// SIMATIC S7-200 project (STEP 7-Micro/WIN), CPU 226 REL 01.01

SYMBOL_TABLE USR1
Any_100ms_Timer  T38
END_SYMBOL_TABLE

SYMBOL_TABLE USS Protocol
USS_LOW_V        VD1000   // (DWORD) Enter the starting address for USS Protocol symbols here.
USS_HIGH_V       VD1004
USS_TIME_OUT     VW1008
USS_I_LINE       VW1010
USS_DAT_PTR0     VD1012
USS_ACT_DRV0     VD1016
USS_CUR_DRV0     VD1020
USS_P0           V1024.0
USS_REQ_SNT0     V1024.1
USS_RETRY_P0     VB1025
USS_ERR_CODE     VB1026
USS_CS_D0        VD1027
USS_CS_W0        VW1027
USS_CS_W2        VW1029
USS_CS_B0        VB1027
USS_CS_B1        VB1028
USS_POLL_BUF     VB1031
USS_XMT_0        VB1046
USS_XMT_ADR0     VB1049
USS_X_STWD       VD1056
USS_X_BCC        VB1060
USS_X_DW1        VD1047
USS_X_DW5        VD1051
USS_X_DW9        VD1055
USS_X_DB13       VB1059
USS_RCV_BUF0     VB1061
USS_R_STX        VB1062
USS_R_LGE        VB1063
USS_R_ADR        VB1064
USS_R_STWD       VD1071
USS_R_DW1        VD1062
USS_R_DW5        VD1066
USS_R_DW9        VD1070
USS_R_W13        VW1074
USS_STAT_TAB     VB1076
USS_ADR_P0       VB1396
END_SYMBOL_TABLE

ORGANIZATION_BLOCK MAIN:OB1
TITLE=在一包装流水线上，设备1是一个负责打包的电机，设备2是一个用于封口的加热器，设备3是一个传送带。操作员通过启动按钮1启动打包电机运行5秒，输出控制在设备1输出，其计时状态记录在计时值1中；按下启动按钮2启动加热器运行8秒，控制设备2输出，计时值2实时更新；按下启动按钮3启动传送带运行10秒，控制设备3输出，计时值3同步记录。设备1、设备2和设备3的运行由各自的启动按钮独立控制，支持同时运行以提高效率。
// 只有当相应的启动按钮被按下时，例如启动按钮1，计时值1才会开始计时并激活设备1输出，确保设备只在需要时运行。设备运行期间，设备1输出会在5秒内保持置位，计时值1实时更新，直到达到预设时间后自动关闭；设备2输出和设备3输出同理分别在8秒和10秒后停止。通过计时值1、计时值2和计时值3配合预定时间，设备能够精确运行并自动关闭。如果生产线需要暂停或出现紧急情况，操作员可以按下复位按钮，此时计时值1、计时值2和计时值3会同时清零，设备1输出、设备2输出和设备3输出也会立即关闭，使系统迅速恢复到初始状态。
// 
BEGIN
Network 1
LD     I0.0
CALL   Timer:SBR0, 50, VW0, Q0.0
Network 2
LD     I0.1
CALL   Timer:SBR0, 80, VW2, Q0.1
Network 3
LD     I0.2
CALL   Timer:SBR0, 100, VW4, Q0.2
Network 4 // Reset network
LD     I0.3
LPS
MOVW   +0, VW0
AENO
MOVW   +0, VW2
AENO
MOVW   +0, VW4
LPP
R      Q0.0, 3
END_ORGANIZATION_BLOCK

SUBROUTINE_BLOCK Timer:SBR0
TITLE=
VAR_INPUT
Timer_PT:WORD;	// LW0 
END_VAR
VAR_IN_OUT
Timer_CV:WORD;	// LW2 
END_VAR
VAR_OUTPUT
Timer_Out:BOOL;	// L4.0 
END_VAR
BEGIN
Network 1 // This example will only work for 100ms timers
LD     SM0.0
MOVW   #Timer_CV:LW2, Any_100ms_Timer:T38
TON    Any_100ms_Timer:T38, #Timer_PT:LW0
MOVW   Any_100ms_Timer:T38, #Timer_CV:LW2
A      Any_100ms_Timer:T38
=      #Timer_Out:L4.0
END_SUBROUTINE_BLOCK
